// TIA Portal V17 export
// export: Created 2026-04-13T11:12:02.810031Z, ExportSetting WithDefaults, DisplayName Totally Integrated Automation Portal, DisplayVersion V17 Update 4, DisplayName TIA Portal Openness, DisplayVersion V17 Update 4, DisplayName TIA Portal Version Control Interface, DisplayVersion V17, DisplayName SINAMICS Startdrive Advanced, DisplayVersion V17, DisplayName SINAMICS Startdrive G130, G150, S120, S150, SINAMICS MV, S210, DisplayVersion V17, DisplayName SINAMICS Startdrive G110M, G120, G120C, G120D, G120P, G115D, DisplayVersion V17, DisplayName STEP 7 Professional, DisplayVersion V17 Update 4, DisplayName STEP 7 Safety, DisplayVersion V17, DisplayName WinCC Professional, DisplayVersion V17 Update 4
ORGANIZATION_BLOCK "Main"   // OB1, SCL, ProgramCycle
TITLE = "Main Program Sweep (Cycle)"
{ S7_Optimized_Access := 'TRUE' }
VERSION : 0.1
// stored: AutoNumber true, IsIECCheckEnabled false, SetENOAutomatically false
   VAR_INPUT
      Initial_Call : Bool;   // Initial call of this OB
      Remanence : Bool;   // =True, if remanent data are available
   END_VAR
BEGIN
   "0- IO Configure"();
   "A1-阀带反馈_DB"();
   "A2-阀带阀导_DB"();
   "A3-电机控制_DB"();
   "A4-脉冲控制_DB"();
   "A6-模拟量输入_DB"();
   "A5-模拟量输出_DB"();
   "A7-温度控制_DB"();
   "6-ALLALARM_DB"();
   "B2--局部连锁_DB"();
   "B3-全局连锁_DB"();
   "B4-清洗连锁_DB"();
   "C1-开式自动_DB"();
   "C2-闭式自动_DB"();
   "C3-室内CIP清洗_DB"();
   "C4-室外CIP清洗_DB"();
   "D1-室内CIP通讯_DB"();
   "D2-室外CIP通讯_DB"();
END_ORGANIZATION_BLOCK
